{attribute addProperty BoxType "EK1122-0000-0018"}
{attribute addProperty Id "Beckhoff_EP8xxxsub_EK1100EK1100_179A0949162A_0001_EP8309_0022_0021EP8309_7EF99CA440851A_0002_EP8309_1022_0016EP8309_7EF99CA440851A_0003_EP8309_1022_0017EP8309_7EF99CA440851A_0004_EP8309_1022_0018EP8309_7EF99CA440851"}
{attribute addProperty CRC "2692164196"}
{attribute addProperty SizeInBites "1648"}
{attribute addProperty SizeInBytes "206"}
TYPE Beckhoff_EP8xxxEK1122_A0772A64 EXTENDS EK1122_179A0949 :
STRUCT
	{attribute addProperty Name "Beckhoff_EP8xxxsub_EK1100"}
	Beckhoff_EP8xxxsub_EK1100 : EK1100_179A0949;
	{attribute addProperty Name "A_0001_EP8309_0022_0021"}
	A_0001_EP8309_0022_0021 : EP8309_7EF99CA4;
	{attribute addProperty Name "A_0002_EP8309_1022_0016"}
	A_0002_EP8309_1022_0016 : EP8309_7EF99CA4;
	{attribute addProperty Name "A_0003_EP8309_1022_0017"}
	A_0003_EP8309_1022_0017 : EP8309_7EF99CA4;
	{attribute addProperty Name "A_0004_EP8309_1022_0018"}
	A_0004_EP8309_1022_0018 : EP8309_7EF99CA4;
END_STRUCT
END_TYPE

(* stored: Version 1.2.0.0, ProductVersion 3.1.4024.9
   DUT Beckhoff_EP8xxxEK1122_A0772A64: Id {dc30b7d7-b645-4e93-a9cc-5e1ceba359f2} *)
